// TIA Portal V17 export
// export: Created 2025-06-26T06:49:21.4330689Z, ExportSetting WithDefaults, DisplayName Totally Integrated Automation Portal, DisplayVersion V17 Update 8, DisplayName TIA Portal Openness, DisplayVersion V17 Update 8, DisplayName TIA Portal Version Control Interface, DisplayVersion V17, DisplayName STEP 7 Professional, DisplayVersion V17 Update 8, DisplayName STEP 7 Safety, DisplayVersion V17 Update 6, DisplayName WinCC Advanced, DisplayVersion V17 Update 8
DATA_BLOCK "Modbus_Master_DB"   // DB38
// stored: AutoNumber true, DBAccessibleFromOPCUA true, InstanceOfName Modbus_Master, OfSystemLibElement Modbus_Master, OfSystemLibVersion 5.0
"Modbus_Master"
   // VAR_INPUT
   //    REQ : Bool;
   //    MB_ADDR : UInt;
   //    MODE : USInt;
   //    DATA_ADDR : UDInt;
   //    DATA_LEN : UInt;
   // END_VAR
   // VAR_OUTPUT
   //    DONE : Bool;
   //    BUSY : Bool;
   //    ERROR : Bool;
   //    STATUS : Word;
   // END_VAR
   // VAR_IN_OUT
   //    DATA_PTR : Variant;
   // END_VAR
   // VAR
   //    MB_State : SInt;
   //    Blocked_Proc_Timeout : Real;
   //    Extended_Addressing : Bool;
   //    Compatibility_Mode : Bool;
   //    MB_DB { S7_SetPoint := 'True'} : P2P_MB_BASE;
   //    Send_P2P { S7_SetPoint := 'True'} : Send_P2P;
   //    Receive_P2P { S7_SetPoint := 'True'} : Receive_P2P;
   //    Receive_Reset { S7_SetPoint := 'True'} : Receive_Reset;
   //    S_PORT : Word;
   //    S_RESP_TO : Word;
   //    S_ICHAR_GAP : Word;
   //    S_RETRIES : Word;
   //    S_MB_ADDR : UInt;
   //    S_MODE : USInt;
   //    S_DATA_ADDR : UDInt;
   //    S_DATA_LEN : UInt;
   //    w_retries : Word;
   //    y_SlaveAddrHi : Byte;
   //    y_SlaveAddrLo : Byte;
   //    StartAddress : Word;
   //    Value : Word;
   //    y_FCode : Byte;
   //    INTERNAL_CDATA : Array[1..257] of Byte;
   //    mb_timer { S7_SetPoint := 'True'} : TON_TIME;
   //    TimeElapsed : Bool;
   // END_VAR
BEGIN
END_DATA_BLOCK
